FUNCTION_BLOCK Test_StringSplitter_ReturnsRemainder EXTENDS TUnitTestBase
VAR
END_VAR

METHOD  Execute
VAR_INST
    StringSplitter : TStringSplitter;
END_VAR
Test_Started();

StringSplitter.Init(
    Str    := 'Bob$TCharles$TDavid',
    Delim1 := '$T',
    Delim2 := '');

Assertion.AssertEquals_BOOL(
    Expected := TRUE,
    Actual   := StringSplitter.HasMore(),
    ObjectName := _TestName,
    VariableName  := 'StringSplitter.HasMore()');
    
Assertion.AssertEquals_STRING(
    Expected := 'Bob',
    Actual   := StringSplitter.GetNext(),
    ObjectName := _TestName,
    VariableName  := 'StringSplitter.GetNext()');
    
Assertion.AssertEquals_STRING(
    Expected := 'Charles$TDavid',
    Actual   := StringSplitter.GetRemainder(),
    ObjectName := _TestName,
    VariableName  := 'StringSplitter.GetRemainder()');

Assertion.AssertEquals_STRING(
    Expected := '',
    Actual   := StringSplitter.GetRemainder(),
    ObjectName := _TestName,
    VariableName  := 'StringSplitter.GetRemainder()');

Assertion.AssertEquals_BOOL(
    Expected := FALSE,
    Actual   := StringSplitter.HasMore(),
    ObjectName := _TestName,
    VariableName  := 'StringSplitter.HasMore()');
    

Test_Finished();
END_METHOD

END_FUNCTION_BLOCK

(* stored: Version 1.1.0.1, ProductVersion 3.1.4024.3
   POU Test_StringSplitter_ReturnsRemainder: Id {8f4fe42a-2bd0-0874-1c8d-73d72a974ba0}, SpecialFunc None
   Method Execute: Id {23d348c2-0106-0a8a-3b8a-b51e96e82332} *)
